FUNCTION_BLOCK FB_Setpoint_Generator
VAR CONSTANT
	nNoOfRows											: INT:= 45;
END_VAR
VAR
	fManValue											: LREAL;
	eMode												: E_CTRL_MODE;
	nSetpointIndex										: INT:= 3;
	fCurrentSetpoint									: LREAL;
	bValueReached										: BOOL;

	fbCTRL_SETPOINT_GENERATOR							: FB_CTRL_SETPOINT_GENERATOR;
	stCTRL_SETPOINT_GENERATOR_PARAMS					: ST_CTRL_SETPOINT_GENERATOR_PARAMS;
	arSetpointTable										: ARRAY [1..nNoOfRows] OF FLOAT;

	eErrorId											: E_CTRL_ERRORCODES;
	bError												: BOOL;

	bInit, bUpdate										: BOOL	:= TRUE;
	fbTON												: TON;
	
	fbGetCurTaskIdx 									: GETCURTASKINDEX;
	bFirstCycle											: BOOL;
	fCycleTime											: LREAL := 0.025;
//	Scope
	fInToScope											: LREAL;
	fOutToScope											: LREAL;
END_VAR

// =========================================================
	// Get task first cycle flag	
fbGetCurTaskIdx(); 
bFirstCycle:= _TaskInfo[fbGetCurTaskIdx.index].FirstCycle;

IF bFirstCycle THEN
	;
END_IF

// Get Cycle Time
IF(GETCURTASKINDEXEX()<=0)THEN
	fCycletime:= TO_LREAL(0.025);(* Don't know, just guessing *)
ELSE
	fCycletime:= UDINT_TO_LREAL(_TaskInfo[GETCURTASKINDEXEX()].cycleTime)/10000000.0;
END_IF

// =========================================================

(*
IF bInit THEN
	(* init the setpoint array *)
	arSetpointTable[ 1 ]	:= 12;
	arSetpointTable[ 2 ]	:= 25;
	arSetpointTable[ 3 ]	:= 42;
	arSetpointTable[ 4 ]	:= 73;

	(* init parameter struct *)
	stCTRL_SETPOINT_GENERATOR_PARAMS.tTaskCycleTime				:= T#10MS;
	stCTRL_SETPOINT_GENERATOR_PARAMS.tCtrlCycleTime				:= T#10MS;
	stCTRL_SETPOINT_GENERATOR_PARAMS.bDisableRamping			:= FALSE;
	stCTRL_SETPOINT_GENERATOR_PARAMS.fVeloNeg					:= 10;
	stCTRL_SETPOINT_GENERATOR_PARAMS.fVeloPos					:= 8;
	stCTRL_SETPOINT_GENERATOR_PARAMS.nDataTable_NumberOfRows	:= 4;

	(* set the mode to ACTIVE --> normal operation *)
	eMode := eCTRL_MODE_ACTIVE;

	(* reset init flag *)
	bInit := FALSE;
END_IF
*)

(*
(* set the addresses *)
stCTRL_SETPOINT_GENERATOR_PARAMS.nDataTable_SIZEOF			:= SIZEOF(arSetpointTable);
stCTRL_SETPOINT_GENERATOR_PARAMS.pDataTable_ADR				:= ADR(arSetpointTable);

(* generate setpoint-index *)
fbTON( IN := TRUE,
		PT	:= T#5s);
IF fbTON.Q
THEN
	nSetpointIndex	:=  nSetpointIndex + 1;
	IF nSetPointIndex > 4
	THEN
		nSetPointIndex := 1;
	END_IF
	fbTON( IN := FALSE);
END_IF


(* copy var to scope var *)
fInToScope := INT_TO_FLOAT(nSetpointIndex);

(* call setpointgenerator *)
fbCTRL_SETPOINT_GENERATOR(	nSetpointIndex		:= nSetpointIndex,
										fManValue				:= fManValue,
										eMode					:= eMode,
										stParams				:= stCTRL_SETPOINT_GENERATOR_PARAMS,
										fOut					=> fCurrentSetpoint,
										bValueReached		=> bValueReached
										 );

(* copy var to scope var *)
fOutToScope := fCurrentSetpoint;
*)

//FB_Init is always available implicitly and it is used primarily for initialization.
//The return value is not evaluated. For a specific influence, you can also declare the
//methods explicitly and provide additional code there with the standard initialization
//code. You can evaluate the return value.
METHOD FB_Init: BOOL
VAR_INPUT
    bInitRetains: BOOL; // TRUE: the retain variables are initialized (reset warm / reset cold)
    bInCopyCode: BOOL;  // TRUE: the instance will be copied to the copy code afterward (online change)   
END_VAR
// =========================================================
(* Init the setpoint array *)
arSetpointTable[ 1 ]	:= 25;
arSetpointTable[ 2 ]	:= 30;
arSetpointTable[ 3 ]	:= 35;
arSetpointTable[ 4 ]	:= 40;
arSetpointTable[ 5 ]	:= 45;
arSetpointTable[ 6 ]	:= 50;
arSetpointTable[ 7 ]	:= 55;
arSetpointTable[ 8 ]	:= 60;
arSetpointTable[ 9 ]	:= 65;
arSetpointTable[ 10 ]	:= 70;
arSetpointTable[ 11 ]	:= 75;
arSetpointTable[ 12 ]	:= 80;
arSetpointTable[ 13 ]	:= 85;
arSetpointTable[ 14 ]	:= 90;
arSetpointTable[ 15 ]	:= 95;
arSetpointTable[ 16 ]	:= 100;
arSetpointTable[ 17 ]	:= 105;
arSetpointTable[ 18 ]	:= 110;
arSetpointTable[ 19 ]	:= 115;
arSetpointTable[ 20 ]	:= 120;
arSetpointTable[ 21 ]	:= 125;
arSetpointTable[ 22 ]	:= 130;
arSetpointTable[ 23 ]	:= 135;
arSetpointTable[ 24 ]	:= 140;
arSetpointTable[ 25 ]	:= 145;
arSetpointTable[ 26 ]	:= 150;
arSetpointTable[ 27 ]	:= 155;
arSetpointTable[ 28 ]	:= 160;
arSetpointTable[ 29 ]	:= 165;
arSetpointTable[ 30 ]	:= 170;
arSetpointTable[ 31 ]	:= 175;
arSetpointTable[ 32 ]	:= 180;
arSetpointTable[ 33 ]	:= 185;
arSetpointTable[ 34 ]	:= 190;
arSetpointTable[ 35 ]	:= 195;
arSetpointTable[ 36 ]	:= 200;
arSetpointTable[ 37 ]	:= 205;
arSetpointTable[ 38 ]	:= 210;
arSetpointTable[ 39 ]	:= 215;
arSetpointTable[ 40 ]	:= 220;
arSetpointTable[ 41 ]	:= 225;
arSetpointTable[ 42 ]	:= 230;
arSetpointTable[ 43 ]	:= 235;
arSetpointTable[ 44 ]	:= 240;
arSetpointTable[ 45 ]	:= 245;

(*
(* Init parameter struct *)
stCTRL_SETPOINT_GENERATOR_PARAMS.tTaskCycleTime				:= UDINT_TO_TIME(_TaskInfo[GETCURTASKINDEXEX()].cycleTime/10000);
stCTRL_SETPOINT_GENERATOR_PARAMS.tCtrlCycleTime				:= UDINT_TO_TIME(_TaskInfo[GETCURTASKINDEXEX()].cycleTime/10000);
stCTRL_SETPOINT_GENERATOR_PARAMS.bDisableRamping			:= FALSE;
stCTRL_SETPOINT_GENERATOR_PARAMS.fVeloNeg					:= 10;
stCTRL_SETPOINT_GENERATOR_PARAMS.fVeloPos					:= 8;
stCTRL_SETPOINT_GENERATOR_PARAMS.nDataTable_NumberOfRows	:= 4;

(* Set the mode to ACTIVE --> normal operation *)
eMode := eCTRL_MODE_ACTIVE;
*)
// =========================================================
END_METHOD

METHOD PUBLIC M_Cyclic
VAR_INPUT
END_VAR
// =========================================================
IF bInit OR bUpdate THEN
	(* Init parameter struct *)
	stCTRL_SETPOINT_GENERATOR_PARAMS.tTaskCycleTime				:= UDINT_TO_TIME(_TaskInfo[GETCURTASKINDEXEX()].cycleTime/10000);
	stCTRL_SETPOINT_GENERATOR_PARAMS.tCtrlCycleTime				:= UDINT_TO_TIME(_TaskInfo[GETCURTASKINDEXEX()].cycleTime/10000);
	stCTRL_SETPOINT_GENERATOR_PARAMS.bDisableRamping			:= FALSE; (*A continuous output value is not calculated if this parameter is TRUE. There is a step change between the output values*)
	stCTRL_SETPOINT_GENERATOR_PARAMS.fVeloNeg					:= 10; (* In units per second *)
	stCTRL_SETPOINT_GENERATOR_PARAMS.fVeloPos					:= 8;  (* In units per second *)
	stCTRL_SETPOINT_GENERATOR_PARAMS.nDataTable_NumberOfRows	:= nNoOfRows;

	(* Set the mode to ACTIVE --> normal operation *)
	eMode := eCTRL_MODE_ACTIVE;
	(* Reset the init flag *)
	bInit := FALSE;
	(* Reset the update flag *)
	bUpdate := FALSE;
END_IF

(* Set the addresses *)
stCTRL_SETPOINT_GENERATOR_PARAMS.nDataTable_SIZEOF			:= SIZEOF(arSetpointTable);
stCTRL_SETPOINT_GENERATOR_PARAMS.pDataTable_ADR				:= ADR(arSetpointTable);

(* Generate setpoint-index *)
fbTON( IN := TRUE, PT:= T#5S);
IF fbTON.Q
THEN
	nSetpointIndex	:=  nSetpointIndex + 1;
	IF nSetPointIndex > 4
	THEN
		nSetPointIndex := 1;
	END_IF
	fbTON( IN := FALSE);
END_IF

(* Copy var to scope var *)
fInToScope := INT_TO_FLOAT(nSetpointIndex);

(* Call setpointgenerator *)
fbCTRL_SETPOINT_GENERATOR(nSetpointIndex:= nSetpointIndex,
										fManValue				:= fManValue,
										eMode					:= eMode,
										stParams				:= stCTRL_SETPOINT_GENERATOR_PARAMS,
										fOut					=> fCurrentSetpoint,
										bValueReached		=> bValueReached
										 );

(* Copy var to scope var *)
fOutToScope := fCurrentSetpoint;

// =========================================================
END_METHOD

END_FUNCTION_BLOCK

(* stored: Version 1.1.0.1
   POU FB_Setpoint_Generator: Id {ba46414f-087c-4b1c-8465-4eeebd5edc8b}, SpecialFunc None
   Method FB_Init: Id {934b235d-9833-48db-b6f4-391752153908}
   Method M_Cyclic: Id {2bbf86ce-9f52-4111-bf2f-dbebf9a0a72b} *)
